{attribute 'qualified_only'}
{attribute 'strict'}
{attribute 'to_string'}
TYPE E_STATION_GEAR_DISTANCE_AXIS :
(
  // which axis nSync distance is checked for termination of GearInPosCA.
  // after nSync distance the station does a regular outfeed to target station
	FOLLOW_THE_MASTER,
  FOLLOW_THE_SLAVE
)UINT;
END_TYPE

(* stored: Version 1.1.0.1, ProductVersion 3.1.4026.18
   DUT E_STATION_GEAR_DISTANCE_AXIS: Id {ca446ba2-2ee4-4f22-b58e-40c69fe43394} *)
